Yaskawa INFORM job: VISUMATIC-FEEDSCREW.JBI

/JOB
//NAME VISUMATIC-FEEDSCREW
//POS
///NPOS 0,0,0,0,0,0
//INST
///DATE 2021/02/04 14:20
///ATTR SC,RW
///GROUP1 RB1
NOP
DOUT OT#(1) ON
END
